PROGRAM main
VAR
	start AT %IX0.0 : bool;
	start_cmd AT %QX0.2 : bool;
	start_coil AT %QX0.1 : bool;
	start_coil0 AT %QX0.2 : bool;
	stop AT %IX0.1 : bool;
	stop_cmd AT %QX0.3 : bool;
	led AT %QX0.0 : bool;
END_VAR

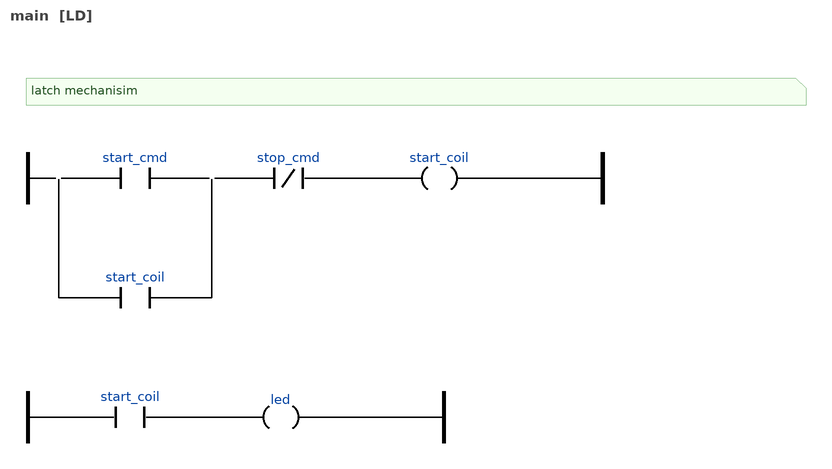
(* LD diagram, written out as Structured Text *)
(* latch mechanisim *)
start_coil := (start_cmd OR start_coil) AND NOT stop_cmd;
led := start_coil;
END_PROGRAM
